TYPE stError_AnalogueInput :
STRUCT
	LowLowAlarm:BOOL 	(*Value below low low set point*)
	HighHighAlarm:BOOL; (*Value above high high set point*)
	Invalid:BOOL; 		(*Invalid input*)
END_STRUCT
END_TYPE

(* stored: Version 1.1.0.1, ProductVersion 3.1.4024.11
   DUT stError_AnalogueInput: Id {80860b6f-e61c-42b0-8546-7e1cad739aa2} *)
